// Mitsubishi GX Works2 project: sequenceEx1   PLC: Q03UDV

PROGRAM MAIN
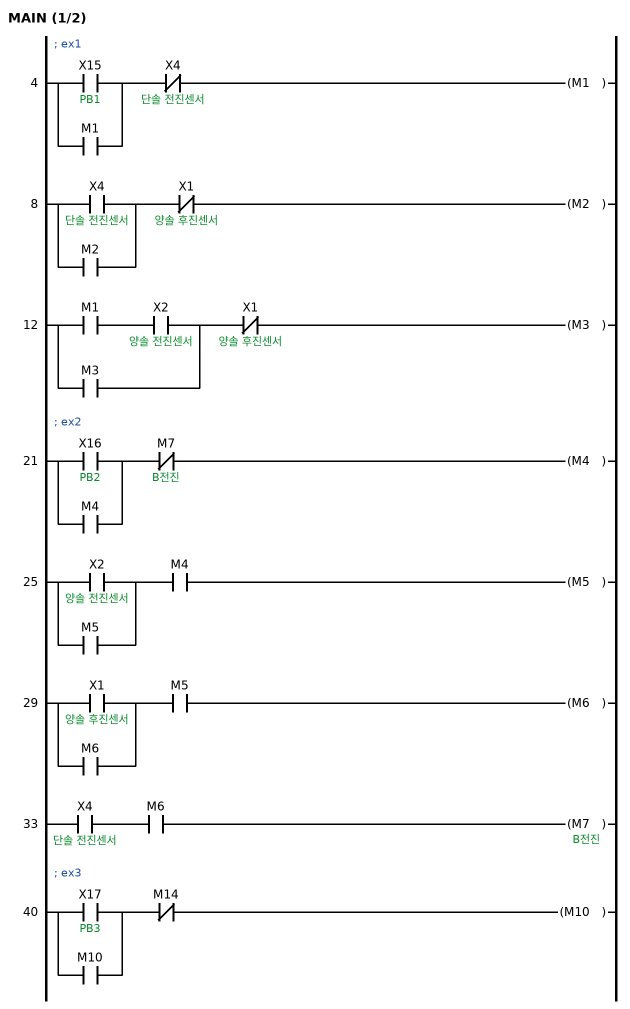
; ex1
4     LD      X15  ; PB1
      OR      M1
      ANI     X4  ; 단솔 전진센서
      OUT     M1
8     LD      X4  ; 단솔 전진센서
      OR      M2
      ANI     X1  ; 양솔 후진센서
      OUT     M2
12    LD      M1
      AND     X2  ; 양솔 전진센서
      OR      M3
      ANI     X1  ; 양솔 후진센서
      OUT     M3
; ex2
21    LD      X16  ; PB2
      OR      M4
      ANI     M7  ; B전진
      OUT     M4
25    LD      X2  ; 양솔 전진센서
      OR      M5
      AND     M4
      OUT     M5
29    LD      X1  ; 양솔 후진센서
      OR      M6
      AND     M5
      OUT     M6
33    LD      X4  ; 단솔 전진센서
      AND     M6
      OUT     M7  ; B전진
; ex3
40    LD      X17  ; PB3
      OR      M10
      ANI     M14
      OUT     M10
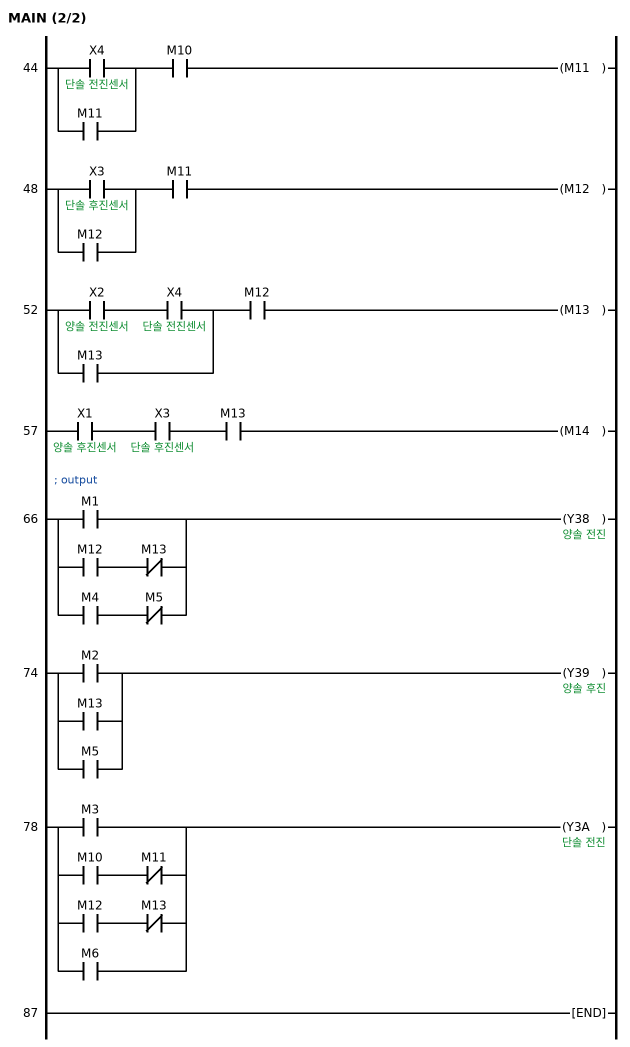
44    LD      X4  ; 단솔 전진센서
      OR      M11
      AND     M10
      OUT     M11
48    LD      X3  ; 단솔 후진센서
      OR      M12
      AND     M11
      OUT     M12
52    LD      X2  ; 양솔 전진센서
      AND     X4  ; 단솔 전진센서
      OR      M13
      AND     M12
      OUT     M13
57    LD      X1  ; 양솔 후진센서
      AND     X3  ; 단솔 후진센서
      AND     M13
      OUT     M14
; output
66    LD      M1
      LD      M12
      ANI     M13
      ORB
      LD      M4
      ANI     M5
      ORB
      OUT     Y38  ; 양솔 전진
74    LD      M2
      OR      M13
      OR      M5
      OUT     Y39  ; 양솔 후진
78    LD      M3
      LD      M10
      ANI     M11
      ORB
      LD      M12
      ANI     M13
      ORB
      OR      M6
      OUT     Y3A  ; 단솔 전진
87    END
END_PROGRAM

// device comments not shown above
M8  ; 둘다 전진
M9  ; 둘다 전진이면
